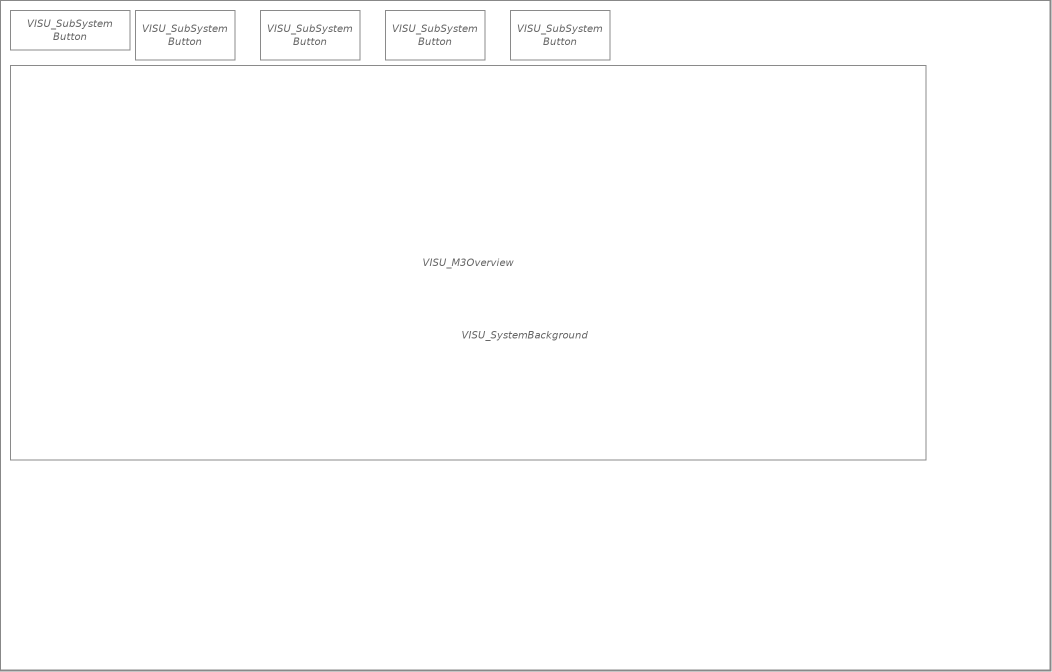
VISUALIZATION VISU_M3  // 1052x672
VAR_IN_OUT
    m3 : M3;
	m3Widget : M3Widget;
END_VAR
    Frame (0,0 1050x670)
        shows VISU_SystemBackground(color := m3Widget.actualStatus.color)
    Frame (10,65 916x395)
        shows VISU_M3Overview(m3 := m3, m3Widget := m3Widget)
        shows VISU_M3Rotation(ref := m3.parts.rotation, widget := m3Widget.rotation, m3Ref := m3, m3Widget := m3Widget)
        shows VISU_M3Translation(ref := m3.parts.translation, widget := m3Widget.translation)
        shows VISU_M3IO(ref := m3.parts.io, widget := m3Widget.io)
        shows VISU_M3Config(m3Widget := m3Widget, editableConfig := m3.editableConfig, activeConfig := m3.config, mgr := m3.parts.configManager, mgrWidget := m3Widget.configManager)
    Frame (10,10 120x40)
        shows VISU_SubSystemButton(widget := m3Widget.button_overview)
        OnMouseClick: FrameSelectionChange Selection=SelectedFrame=f0c0c79d-59b2-407d-9a73-98e777c3e69e, GlobSel=AssignType=Directly, SelType=Locally
        OnMouseClick: execute { m3Widget.activeTab := M3Tabs.OVERVIEW; }
    Frame (135,10 100x50)
        shows VISU_SubSystemButton(widget := m3Widget.button_rotation)
        OnMouseClick: FrameSelectionChange Selection=SelectedFrame=f0c0c79d-59b2-407d-9a73-98e777c3e69e, Selection=1, GlobSel=AssignType=Directly, SelType=Locally
        OnMouseClick: execute { m3Widget.activeTab := M3Tabs.ROTATION; }
    Frame (260,10 100x50)
        shows VISU_SubSystemButton(widget := m3Widget.button_translation)
        OnMouseClick: FrameSelectionChange Selection=SelectedFrame=f0c0c79d-59b2-407d-9a73-98e777c3e69e, Selection=2, GlobSel=AssignType=Directly, SelType=Locally
        OnMouseClick: execute { m3Widget.activeTab := M3Tabs.TRANSLATION; }
    Frame (385,10 100x50)
        shows VISU_SubSystemButton(widget := m3Widget.button_io)
        OnMouseClick: FrameSelectionChange Selection=SelectedFrame=f0c0c79d-59b2-407d-9a73-98e777c3e69e, Selection=3, GlobSel=AssignType=Directly, SelType=Locally
        OnMouseClick: execute { m3Widget.activeTab := M3Tabs.IO; }
    Frame (510,10 100x50)
        shows VISU_SubSystemButton(widget := m3Widget.button_config)
        OnMouseClick: FrameSelectionChange Selection=SelectedFrame=f0c0c79d-59b2-407d-9a73-98e777c3e69e, Selection=4, GlobSel=AssignType=Directly, SelType=Locally
        OnMouseClick: execute { m3Widget.activeTab := M3Tabs.CONFIG; }
END_VISUALIZATION

(* stored: Version 1.1.0.1, ProductVersion 3.1.4019.2
   Visu VISU_M3: Id {7b000a81-8f4d-4a12-87cd-3fda77383a07} *)
